FUNCTION_BLOCK ABSTRACT FBA_LinearTrifecta EXTENDS FBA_LinearDrive
VAR
	outerLimit AT %I* : BOOL;
END_VAR
(*
this abstract FB adds a rear limit sensor to FBA_Drive
*)

{attribute 'monitoring':='call'}
PROPERTY AtOuterLimit : BOOL
GET
AtOuterLimit := outerLimit <> limitSensorDefaultState;
END_GET
END_PROPERTY

END_FUNCTION_BLOCK

(* stored: Version 1.1.0.1, ProductVersion 3.1.4024.11
   POU FBA_LinearTrifecta: Id {983d112e-9036-4684-9de5-17676cefe2c2}, SpecialFunc None
   Property AtOuterLimit: Id {dac0e275-c238-4d97-9eb5-b53ff5d109b5}
   Get Get: Id {8e2cf29f-baab-4478-a786-49db2b481578} *)
